// TIA Portal V18 export
// export: Created 2025-12-01T17:51:17.7499704Z, ExportSetting None, DisplayName Totally Integrated Automation Portal, DisplayVersion V18 Update 5, DisplayName TIA Portal Openness, DisplayVersion V18 Update 5, DisplayName TIA Portal Teamcenter Gateway, DisplayVersion V18, DisplayName TIA Portal Version Control Interface, DisplayVersion V18, DisplayName STEP 7 Professional, DisplayVersion V18 Update 5, DisplayName STEP 7 Safety, DisplayVersion V18, DisplayName WinCC Professional, DisplayVersion V18 Update 5
FUNCTION "Servo" : Void   // FC2500, LAD
{ S7_Optimized_Access := 'TRUE' }
// stored: AutoNumber false, SetENOAutomatically false
BEGIN

REGION Network 1
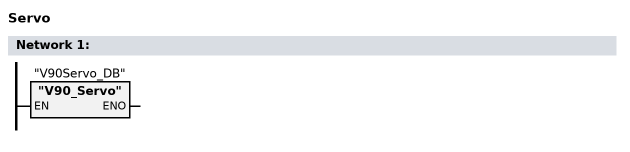
   RUNG wire#powerrail
      "V90Servo_DB"()
   END_RUNG
   // the same network as SCL:
   "V90Servo_DB"();   // "V90_Servo"
END_REGION
END_FUNCTION
